Yaskawa INFORM job: INIT_ROS.JBI

/JOB
//NAME INIT_ROS
//POS
///NPOS 0,0,0,0,0,0
//INST
///DATE 2013/03/29 05:32
///ATTR SC,RW
///GROUP1 RB1
NOP
IF ( IN#(1871)=ON AND IN#(1872)=OFF ) THEN
 CALL JOB:MAIN
ENDIF
DOUT OT#(890) OFF
DOUT OT#(889) OFF
TIMER T=0.05
DOUT OT#(889) ON //ROS_READY
WAIT OT#(890)=ON //ROS_DONE
DOUT OT#(890) OFF
END
